// TIA Portal V17 export
// export: Created 2025-06-26T07:49:17.9307778Z, ExportSetting WithDefaults, DisplayName Totally Integrated Automation Portal, DisplayVersion V17 Update 8, DisplayName TIA Portal Openness, DisplayVersion V17 Update 8, DisplayName TIA Portal Version Control Interface, DisplayVersion V17, DisplayName STEP 7 Professional, DisplayVersion V17 Update 8, DisplayName STEP 7 Safety, DisplayVersion V17 Update 6, DisplayName WinCC Advanced, DisplayVersion V17 Update 8
DATA_BLOCK "DB_System"   // DB42
{ S7_Optimized_Access := 'TRUE' }
VERSION : 0.1
// stored: AutoNumber false, DBAccessibleFromOPCUA true, IsOnlyStoredInLoadMemory false, IsRetainMemResEnabled false, IsWriteProtectedInAS false, MemoryReserve 100
   VAR
      bFirstCycle : Bool := FALSE;   // High on first scan only
      bFirstCycleCyclic : Bool := FALSE;
      bSimulation : Bool := FALSE;   // Simulation active
      SoftwareVersion : String := 'V4.0.0.7';   // PLC software version string
      S7CommEnable : Bool := true;   // Do S7 comm with Process PLC
   END_VAR
   VAR RETAIN
      ClientID : String := 'default';   // used by MQTT
   END_VAR
BEGIN
END_DATA_BLOCK
